TYPE ST_Configuration :
STRUCT
  XtsStationParameter  : ARRAY[1..MAX_STATION] OF ST_STATION_PARAMETER;
END_STRUCT
END_TYPE

(* stored: Version 1.1.0.1, ProductVersion 3.1.4026.18
   DUT ST_Configuration: Id {1a6e1536-77e9-4793-aea9-2b95e9d3473a} *)
